Staubli VAL3: remGetHeartbeat.pgx

program remGetHeartbeat(string& sReturn[] (dimensions=1))
  local string sCmd
begin
  // Return the PPS status saved in the robot
  //
  logMsg("call remGetHeartBeat")
  sCmd="GETHEARTBEAT"
  call remGetnGlobal(nHeartbeat,sCmd,sReturn)
end
